# EPICS substitutions: db/ecmcEL3702_s100.substitutions
file ecmcEcSlave.template
{
    pattern {}
            {}
}

file ecmcEL3702-chX.template
{
	pattern {CH_ID, DTYP,             FTVL,  NELM }
		    {1,     asynInt16ArrayIn, SHORT, 100  }
		    {2,     asynInt16ArrayIn, SHORT, 100  }
}
